TYPE TFMachinePalletizer_ModuleState :
STRUCT
	Cmd	  : UDINT;
	CmdCase : UDINT;
	Error : UDINT;
	ErrorExtra : UDINT;
END_STRUCT
END_TYPE

(* stored: Version 1.1.0.1, ProductVersion 3.1.4024.11
   DUT TFMachinePalletizer_ModuleState: Id {b36a8a4a-f578-44aa-b0d8-90a27b91d5ad} *)
